FUNCTION_BLOCK FB_SaMElementUnHolding EXTENDS FB_SaMElement
VAR
END_VAR

END_FUNCTION_BLOCK

(* stored: Version 1.1.0.1
   POU FB_SaMElementUnHolding: Id {f512916e-13a4-02a1-381c-98ad00edcef5}, SpecialFunc None *)
